PROGRAM PRG_PLC_tasks
VAR
    // variables for testing
    axis: AXIS_REF;
    power: MC_POWER;

    retractedLS AT %I* : BOOL;
    extendedLS At %I* :BOOL;

END_VAR


(*
   This is to test axis safely by both limit switch enabled.
   manually link the variables "retractedLS" and "extendedLS" to the imit switches inputs

   Standard limit switches are NC, enable/disable both directions directly by limit switches
  if limit swithes are NO, enable/disable the related direction using reversed limit switch reading.

*)
power(Axis:=axis, Enable_Positive := retractedLS and extendedLS, Enable_Negative:= extendedLS and retractedLS);
//power(Axis:=axis, Enable_Positive := NOT retractedLS, Enable_Negative:= NOT extendedLS);

PRG_GasNozzleXYZ();
PRG_MainChamber();
PRG_GasJetPointing();
PRG_CoilMovers();
// PRG_SMARACT();

END_PROGRAM

(* stored: Version 1.1.0.1
   POU PRG_PLC_tasks: Id {ed295dcb-e9ae-41f5-8c35-f2cb9f5cb69e}, SpecialFunc None *)
